// TIA Portal V20 export
DATA_BLOCK "RealDbName"   // DB7
   VAR
      Outer { S7_SetPoint := 'True'} : "OuterType";
   END_VAR
BEGIN
END_DATA_BLOCK
